(* IEC 61131-3 sources: Kur_TemplateProject_v1/TestPanelV1.fbsproj/MyController.device.xml.v3^/Plc Logic.plclogic.xml.v3^/Application.application.xml.v3^/Kur_Library/02_Blocks/AlarmSystem.fb.st^, 1 file *)

(* ---- Chk.meth.st ---- *)
METHOD PUBLIC  Chk
VAR_INPUT
    ID      : UINT;
    Alarm   : BOOL;
END_VAR

IF (ID < 1) OR (ID > 100) THEN
    RETURN;
END_IF

Cond[ID] := Alarm;

IF Alarm AND NOT Latch[ID] THEN
    Latch[ID] := TRUE;
    BuzzerLtc := TRUE;
END_IF
